Staubli VAL3: PULSE.pjx

--- PULSE.pjx ---
Parameters version=s7.5 stackSize=5000 millimeterUnit=true
Program file=execute.pgx
Program file=find.pgx
Program file=get.pgx
Program file=getSize.pgx
Program file=getType.pgx
Program file=load.pgx
Program file=onEdit.pgx
Program file=onInsert.pgx
Program file=onProgEnd.pgx
Program file=onRun.pgx
Program file=onStart.pgx
Program file=onStop.pgx
Data file=PULSE.dtx
Library alias=cycleStatus path=Disk://cycleStatus/cycleStatus.pjx
Library alias=out path=Disk://instruction/inputOutput/OUT/OUT.pjx
Library alias=use path=Disk://kernel/userPage/userPage.pjx
Library alias=language path=Disk://kernel/language/language.pjx

--- PULSE.dtx ---
public string sItems[2]
string sMessage
bool bExecute[3]
public string sItemsCycle

--- execute.pgx ---
program execute(string x_sItem, bool& x_bDone[])
  local num l_nValue
  local string l_sItem
  local bool l_bOk
begin
  // compose the string
  call use:stringToArray(x_sItem,sItemsCycle)
  //
  l_bOk=true
  toNum(sItemsCycle[1],l_nValue,l_bOk)
  l_sItem=right(sItemsCycle,len(sItemsCycle)-len("OUT "))
  call out:onRun(l_sItem)
  x_bDone=true
  //
  delay(l_nValue)
  // compose the output to OFF
  l_sItem=left(l_sItem,len(l_sItem)-len(">ON"))+">OFF"
  //
  call out:onRun(l_sItem)
  x_bDone=false
end

--- find.pgx ---
public program find(string& x_sItem[], bool& x_bFound[])
begin
  // search the item in the output
end

--- getSize.pgx ---
public program getSize(num& x_nSize[])
begin
  // how many items
  call out:getSize(x_nSize)
end

--- onEdit.pgx ---
public program onEdit(string& x_sItem[])
  local string l_sItem
  local num l_nValue
  local string l_sType
  local bool l_bOk
begin
  //
  // compose the string
  call use:stringToArray(x_sItem,sItems)
  call getType(l_sType)
  //
  l_bOk=true
  toNum(sItems[1],l_nValue,l_bOk)
  // change the field
  call use:insertDialog(l_sType+" "+x_sItem+"#"+"DELAY [Sec] ",l_nValue,0,100)
  // give back
  x_sItem=sItems+","+toString(".2,",l_nValue)
end

--- onInsert.pgx ---
public program onInsert(string& x_sItem[])
  local num l_nSize
  local num i
  local num l_nKey
  local string l_sMessage
  local string l_sItem
  local bool l_bActive
  local num l_nIndex
  local string l_sType
  local num l_nSizeList
  local num l_nValue
  local string l_sName
  local string l_sItemList
begin
  cls()
  x_sItem=""
  call getSize(l_nSizeList)
  l_nSize=0
  //
  // create the list
  //
  call use:setSizeList(10,0,28,11)
  call use:listcreate("OUTPUT ")
  // insert in the list
  for i=0 to l_nSizeList-1
    call out:get(l_sItem,i)
    call out:isActive(l_bActive,l_sItem)
    if l_bActive
      // insert into the list
      call out:getItem(l_sName,l_sItem)
      l_sItemList=l_sItem+" {"+l_sName+"}"
      call use:listadd(l_sItemList)
    endIf
  endFor
  call use:listredraw(min(l_nIndex-use:nView,0))
  // display the actual item
  call getType(l_sType)
  l_sItem=l_sType
  call use:clear(0,13)
  call language:message(l_sMessage,63)
  call use:typeCenter(13,l_sMessage,40,false)
  do
    l_nKey=get()
    // get one output from the list
    call use:listevent(l_nKey,l_nIndex,l_sItem)
    if l_nKey==255
      return
    endIf
  until l_nKey==270
  // insert the pulse
  call use:insertDialog("DELAY [Sec] ",l_nValue,0,100)
  if !use:bUseEscape
    //
    // insert the sentence
    //
    if l_sItem==""
      return
    else
      l_sItem=left(l_sItem,find(l_sItem,"{")-1)
    endIf
    // return the value
    x_sItem="OUT "+l_sItem+">ON,"+toString(".2",l_nValue)
  endIf
end

--- onRun.pgx ---
public program onRun(string& x_sItem[])
  local bool l_bDone
  local string l_sItem
begin
  //
  // show the string
  //
  do
    if taskStatus("PULSE")==-1
      taskCreate "PULSE",20,execute(x_sItem,bExecute)
      watch(bExecute,0.5)
      l_bDone=true
    elseIf taskStatus("PULSE2")==-1
      taskCreate "PULSE2",20,execute(x_sItem,bExecute[1])
      watch(bExecute[1],0.5)
      l_bDone=true
    elseIf taskStatus("PULSE3")==-1
      taskCreate "PULSE3",20,execute(x_sItem,bExecute[2])
      watch(bExecute[2],0.5)
      l_bDone=true
    endIf
    delay(0)
  until l_bDone==true
end

--- onStop.pgx ---
public program onStop(string& x_sItem[])
  local num i
begin
  // reset the bit
  for i=0 to size(bExecute)-1
    bExecute[i]=false
  endFor
end
